% RSLogix 500 project Resfriador_oleo_bancada.RSS, saved by version 8.40.00.08 %
PROJECT "UNTITLED"    % processor: Bul.1763 MicroLogix 1100 Series B %

PROGRAM FILES
  LAD 2 "PRINCIPAL"  5 rungs
  LAD 3 "COM_BOMB"  3 rungs  % comando liga bomba de oleo %
  LAD 4 "COM_VENT"  2 rungs  % comando para ligar vent %
  LAD 5 "COM_COMP"  2 rungs  % comando para ligar compressor %
  LAD 6 "ALARMS"  2 rungs  % alarmes e reset %

DATA FILES
  O0 OUTPUT  4 elements
  I1 INPUT  6 elements
  S2 STATUS  66 elements
  B3 BINARY  1 elements
  T4 TIMER  1 elements
  C5 COUNTER  1 elements
  R6 CONTROL  1 elements
  N7 INTEGER  1 elements
  F8 FLOAT  1 elements

LADDER 2 "PRINCIPAL"
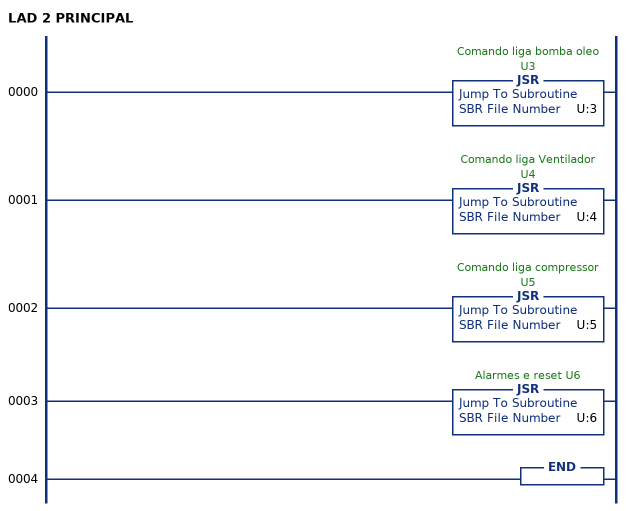
% Rung: 0 %
SOR JSR U:3 EOR
%   U:3  U3  "Comando liga bomba oleo" %
% Rung: 1 %
SOR JSR U:4 EOR
%   U:4  U4  "Comando liga Ventilador" %
% Rung: 2 %
SOR JSR U:5 EOR
%   U:5  U5  "Comando liga compressor" %
% Rung: 3 %
SOR JSR U:6 EOR
%   U:6  U6  "Alarmes e reset" %
% Rung: 4 %
SOR END EOR

LADDER 3 "COM_BOMB"    % comando liga bomba de oleo %
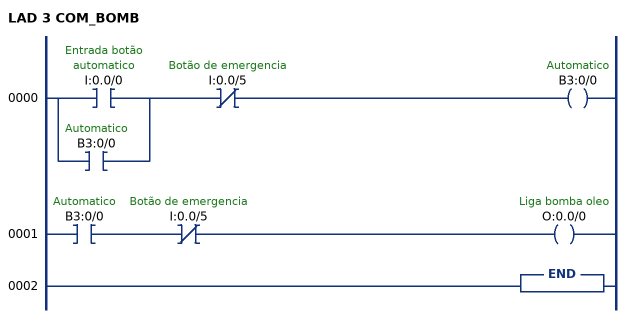
% Rung: 0 %
SOR BST XIC I:0.0/0 NXB XIC B3:0/0 BND XIO I:0.0/5 OTE B3:0/0 EOR
%   I:0.0/0  "Entrada botão automatico" %
%   B3:0/0  "Automatico" %
%   I:0.0/5  "Botão de emergencia" %
% Rung: 1 %
SOR XIC B3:0/0 XIO I:0.0/5 OTE O:0.0/0 EOR
%   B3:0/0  "Automatico" %
%   I:0.0/5  "Botão de emergencia" %
%   O:0.0/0  "Liga bomba oleo" %
% Rung: 2 %
SOR END EOR

LADDER 4 "COM_VENT"    % comando para ligar vent %
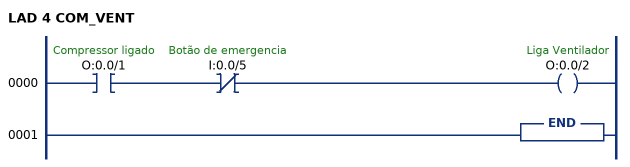
% Rung: 0 %
SOR XIC O:0.0/1 XIO I:0.0/5 OTE O:0.0/2 EOR
%   O:0.0/1  "Compressor ligado" %
%   I:0.0/5  "Botão de emergencia" %
%   O:0.0/2  "Liga Ventilador" %
% Rung: 1 %
SOR END EOR

LADDER 5 "COM_COMP"    % comando para ligar compressor %
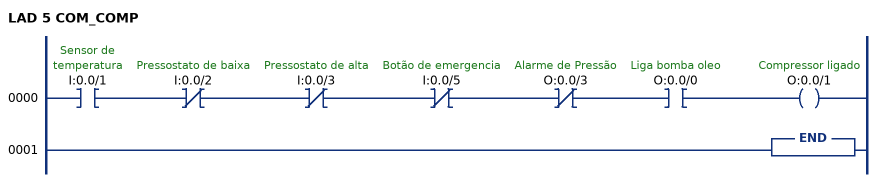
% Rung: 0 %
SOR XIC I:0.0/1 XIO I:0.0/2 XIO I:0.0/3 XIO I:0.0/5 XIO O:0.0/3 XIC O:0.0/0 OTE O:0.0/1 EOR
%   I:0.0/1  "Sensor de temperatura" %
%   I:0.0/2  "Pressostato de baixa" %
%   I:0.0/3  "Pressostato de alta" %
%   I:0.0/5  "Botão de emergencia" %
%   O:0.0/3  "Alarme de Pressão" %
%   O:0.0/0  "Liga bomba oleo" %
%   O:0.0/1  "Compressor ligado" %
% Rung: 1 %
SOR END EOR

LADDER 6 "ALARMS"    % alarmes e reset %
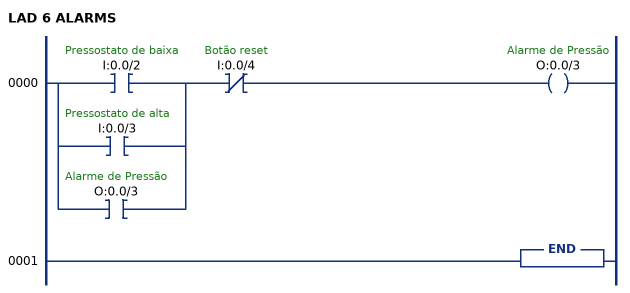
% Rung: 0 %
SOR BST XIC I:0.0/2 NXB BST XIC I:0.0/3 NXB XIC O:0.0/3 BND BND XIO I:0.0/4 OTE O:0.0/3 EOR
%   I:0.0/2  "Pressostato de baixa" %
%   I:0.0/3  "Pressostato de alta" %
%   O:0.0/3  "Alarme de Pressão" %
%   I:0.0/4  "Botão reset" %
% Rung: 1 %
SOR END EOR

OTHER DOCUMENTED ADDRESSES
  B3:0/1  "Liga motor"
  I:0.0  "Automatico/ Manual"
  I:0.1  "Sensor temperatura"
  I:0.1/0  "Setpoint temperatura"
  I:0.2  "Pressostato de baixa"
  I:0.2/0  "Pressostato de baixa"
  I:0.3  "Pressostato de alta"
  I:0.3/0  "Pressostato de alta"
  I:0.4/0  "Botão reset"
  I:0.5  "Emergencia"
  I:0.5/0  "Emergencia"
  I:3  "Pressostato de alta"
  O:0.0  "Liga bomba de oleo"
  O:0.1  "Liga compressor"
  O:0.1/0  "Compressor ligado"
  O:0.2  "Liga ventilador"
  O:0.2/0  "Liga ventilador"
  O:0.3/0  "Alarme de pressão"
  O:0.10  "Liga compressor"
  O:0.10/0  "Liga compressor"
